
        DATA_BLOCK "LabelData"
        { S7_Optimized_Access := 'TRUE' }
        VERSION : 0.1
        NON_RETAIN
        VAR
            TemplateString : WString[1000];
            PlaceHolders : Array[0..5] of Struct
                Id : Int;   // Placeholder ID (0..9)
                Position : Int;   // Startposition in template string
            END_STRUCT;
        END_VAR

        BEGIN
            TemplateString := WSTRING#'^XA^BY2,3,80^FX*Auftrag^FO420,200^A0R,75^FD$${0}^FS^FO420,1000^BCR,,N^FD$${0}^FS^FX*Anzahl^FO320,200^A0R,50^FD$${1} Stk^FS^FX*Datum^FO320,1000^A0R,45^FD$${2}^FS^FX*Type^FO120,200^A0R,45^FD$${3} FDR-1100J^FS^FO120,1000^BCR,,N^FD$${3}^FS^XZ';

            PlaceHolders[0].Id := 0;
            PlaceHolders[0].Position := 43;

            PlaceHolders[1].Id := 0;
            PlaceHolders[1].Position := 71;

            PlaceHolders[2].Id := 1;
            PlaceHolders[2].Position := 108;

            PlaceHolders[3].Id := 2;
            PlaceHolders[3].Position := 149;

            PlaceHolders[4].Id := 3;
            PlaceHolders[4].Position := 184;

            PlaceHolders[5].Id := 3;
            PlaceHolders[5].Position := 222;
        END_DATA_BLOCK